// TIA Portal V20 export
TYPE "TypeSensor"
   STRUCT
      sen : Bool;
      onDel : Bool;
      offDel : Bool;
      occ : Bool;
      occPe : Bool;
      occNe : Bool;
      off : Bool;
      full : Bool;
      free : Bool;
      empty : Bool;
      err : Bool;
      errOcc : Bool;   // fault sensor was to long occupied, maybe dirty or misaligned
      errFree : Bool;   // fault sensor was to long free, maybe dirty or misaligned
      errCycle : Bool;   // fault sensor plausibility check of cycles, after a certain amount(#errCycleVal) of trigger(#errCycleIn) the sensor had no rising or falling edge
      war : Bool;
      refMode : Bool;   // reference mode
      refRun : Bool;   // reference running
      onCntr : Real;   // counter for on delayed
      offCntr : Real;   // counter for off delayed
      occOnCntr : Real;   // on counter for occupied
      occOffCntr : Real;   // on counter for occupied
      val : Real;   // value from sensor, if ex. the sensor is read as a analog input
      occGap : Real;   // gap since last occupied
      "name" : WString[30];   // name, used for fault messages
      description : WString[90];   // description, used for fault messages
   END_STRUCT;
END_TYPE
